TYPE ST_AteqEcho :
STRUCT
	
    (* Byte 0 - 00h *)
    bReset                 : BOOL; // Bit 0
    bStart                 : BOOL; // Bit 1
    bSpecialCycle          : BOOL; // Bit 2
    bProgramSelect         : BOOL; // Bit 3
    bReadFifo              : BOOL; // Bit 4
    bReadParams            : BOOL; // Bit 5
    bWriteParams           : BOOL; // Bit 6
    bResetFifo             : BOOL; // Bit 7

    (* Byte 1 - 01h *)
    bReadConfig            : BOOL; // Bit 0
    bReadExtMenu           : BOOL; // Bit 1
    bReadFunctionBits      : BOOL; // Bit 2
    bWriteExtMenu          : BOOL; // Bit 3
    bWriteFunctionBits     : BOOL; // Bit 4
    bReadProgramName       : BOOL; // Bit 5
    bWriteProgramName      : BOOL; // Bit 6
    bReadLastResult        : BOOL; // Bit 7
	
END_STRUCT
END_TYPE

(* stored: Version 1.1.0.1, ProductVersion 3.1.4024.15
   DUT ST_AteqEcho: Id {80c41e36-cd47-4d38-b0ee-934383f0bb01} *)
